FUNCTION J_Make_Message : STRING
VAR_INPUT
	Operation_Mode : E_Mode_of_operation;
	Testing_Mode   : J_E_Stop_Modes;
	Desired_Value  : DINT;
	Real_Value     : DINT;
	Ranking 	   : J_E_Test_Ranking;
	Comment		   : STRING(256);
END_VAR
VAR
	Message : STRING;
END_VAR

Message := CONCAT(Message, TO_STRING(Operation_Mode));
Message := CONCAT(Message,',');
//Message := CONCAT(Message,'$T');
Message := CONCAT(Message, TO_STRING(Testing_Mode));
Message := CONCAT(Message,',');
//Message := CONCAT(Message,'$T');
Message := CONCAT(Message, DINT_TO_STRING(Desired_Value));
Message := CONCAT(Message,',');
//Message := CONCAT(Message,'$T');
Message := CONCAT(Message, DINT_TO_STRING(Real_Value));
Message := CONCAT(Message,',');
//Message := CONCAT(Message,'$T');
Message := CONCAT(Message, TO_STRING(Ranking));
Message := CONCAT(Message,',');
//Message := CONCAT(Message,'$T');
Message := CONCAT(Message, Comment);
Message := CONCAT(Message,'$n');

GLB.Logger.SaveFlag := TRUE;

J_Make_Message := Message;

END_FUNCTION

(* stored: Version 1.1.0.1, ProductVersion 3.1.4024.12
   POU J_Make_Message: Id {fca63597-66d2-4877-b13d-15141e1310bf}, SpecialFunc None *)
